// TIA Portal V19 export
VAR_GLOBAL   // PLC tag table "Default tag table"
   Tag_1 AT %M1.0 : Bool;
   Tag_2 AT %Q2.0 : Bool;
   Tag_3 AT %M22.0 : Bool;
   Tag_4 AT %Q21.0 : Bool;
   Tag_5 AT %M83.0 : Bool;
   Tag_6 AT %M81.2 : Bool;
   Tag_7 AT %M100.3 : Bool;
   Tag_8 AT %M62.6 : Bool;
   Tag_9 AT %M2001.0 : Bool;
   Tag_10 AT %M21.4 : Bool;
END_VAR
